{attribute 'qualified_only'}
VAR_GLOBAL
	ACK AT%I*:BOOL;	

	dIn_1 AT%I*:BOOL;
	dIn_2 AT%I*:BOOL;
	dIn_3 AT%I*:BOOL;
	dIn_4 AT%I*:BOOL;
	
	dOut_1 AT%Q*:BOOL;
	dOut_2 AT%Q*:BOOL;
	dOut_3 AT%Q*:BOOL;
	dOut_4 AT%Q*:BOOL;
	
	
END_VAR

(* stored: Version 1.1.0.1, ProductVersion 3.1.4022.17
   GVL GVL_IO: Id {5e477ad3-5b10-4379-bbc4-64f19b8a5a3f} *)
